FUNCTION_BLOCK EmitterController
VAR_INPUT
	AtBufferEntry : BOOL;
END_VAR
VAR_OUTPUT
	Emitter : BOOL;
END_VAR
VAR
	TimerTON1 : TON;
	TimerTOF1 : TOF; 
END_VAR

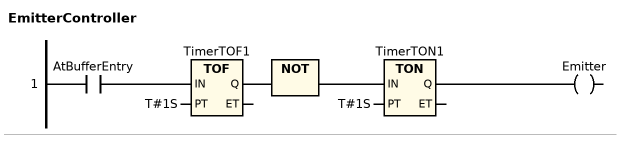
// NETWORK 1
TimerTOF1(IN := AtBufferEntry, PT := T#1S); // TOF
TimerTON1(IN := NOT TimerTOF1.Q, PT := T#1S); // TON
Emitter := TimerTON1.Q;

END_FUNCTION_BLOCK

(* stored: Version 1.1.0.1, ProductVersion 3.1.4024.12
   POU EmitterController: Id {4c700612-52c2-4f11-b50a-ea7e3354bdfb}, SpecialFunc None *)
